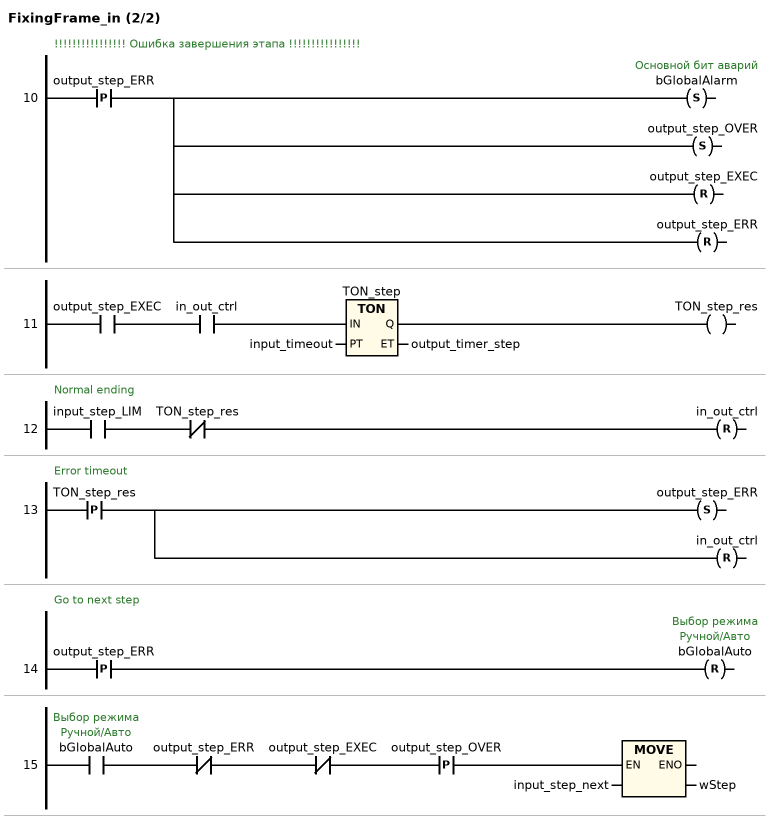
// NETWORK 10
// !!!!!!!!!!!!!!!! Ошибка завершения этапа !!!!!!!!!!!!!!!!
//   bGlobalAlarm: Основной бит аварий
_rt4(CLK := output_step_ERR);
bGlobalAlarm S= _rt4.Q;
output_step_OVER S= _rt4.Q;
output_step_EXEC R= _rt4.Q;
output_step_ERR R= _rt4.Q;

// NETWORK 11
TON_step(IN := output_step_EXEC AND in_out_ctrl, PT := input_timeout, ET => output_timer_step); // TON
TON_step_res := TON_step.Q;

// NETWORK 12
// Normal ending
in_out_ctrl R= input_step_LIM AND NOT TON_step_res;

// NETWORK 13
// Error timeout
_rt5(CLK := TON_step_res);
output_step_ERR S= _rt5.Q;
in_out_ctrl R= _rt5.Q;

// NETWORK 14
// Go to next step
//   bGlobalAuto: Выбор режима Ручной/Авто
_rt6(CLK := output_step_ERR);
bGlobalAuto R= _rt6.Q;

// NETWORK 15
//   bGlobalAuto: Выбор режима Ручной/Авто
_rt7(CLK := output_step_OVER);
IF bGlobalAuto AND NOT output_step_ERR AND NOT output_step_EXEC AND _rt7.Q THEN wStep := input_step_next; END_IF

END_PROGRAM

// MyController/Application/module_unites/FixingFrame_out
PROGRAM FixingFrame_out
VAR_INPUT
	input_step_INIT: BOOL;
	input_step_num: INT;
	input_step_LIM: BOOL;
	input_step_next: INT;
	input_timeout: TIME;
END_VAR

VAR_OUTPUT
	output_step_EXEC: BOOL;
	output_step_OVER: BOOL;
	output_step_ERR: BOOL;
	output_timer_step: TIME;
END_VAR
VAR_IN_OUT
	in_out_ctrl: BOOL;
END_VAR
VAR
	TON_step: TON;
	TON_step_res: BOOL;
	step_active: BOOL;
	TON_delay: TON;
	timer_delay: TIME;
	ton_delay_ok: BOOL;
END_VAR
VAR // added by the converter: edge detectors and wires of the graphical bodies
    _rt1, _rt2, _rt3, _rt4, _rt5, _rt6, _rt7 : R_TRIG;
    _w1, _w2 : BOOL;
    _ft1 : F_TRIG;
END_VAR

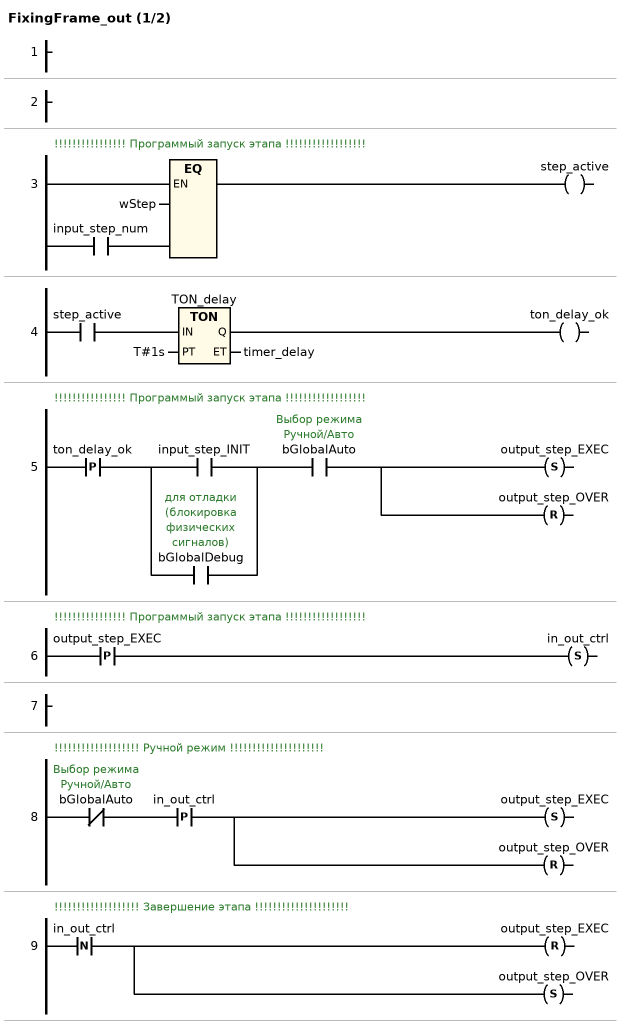
// NETWORK 1

// NETWORK 2

// NETWORK 3
// !!!!!!!!!!!!!!!! Программый запуск этапа !!!!!!!!!!!!!!!!!!
step_active := wStep = input_step_num;

// NETWORK 4
TON_delay(IN := step_active, PT := T#1s, ET => timer_delay); // TON
ton_delay_ok := TON_delay.Q;

// NETWORK 5
// !!!!!!!!!!!!!!!! Программый запуск этапа !!!!!!!!!!!!!!!!!!
//   bGlobalDebug: для отладки (блокировка физических сигналов)
//   bGlobalAuto: Выбор режима Ручной/Авто
_rt1(CLK := ton_delay_ok);
_w1 := _rt1.Q AND (input_step_INIT OR bGlobalDebug) AND bGlobalAuto;
output_step_EXEC S= _w1;
output_step_OVER R= _w1;

// NETWORK 6
// !!!!!!!!!!!!!!!! Программый запуск этапа !!!!!!!!!!!!!!!!!!
_rt2(CLK := output_step_EXEC);
in_out_ctrl S= _rt2.Q;

// NETWORK 7

// NETWORK 8
// !!!!!!!!!!!!!!!!!!! Ручной режим !!!!!!!!!!!!!!!!!!!!!
//   bGlobalAuto: Выбор режима Ручной/Авто
_rt3(CLK := in_out_ctrl);
_w2 := NOT bGlobalAuto AND _rt3.Q;
output_step_EXEC S= _w2;
output_step_OVER R= _w2;

// NETWORK 9
// !!!!!!!!!!!!!!!!!!! Завершение этапа !!!!!!!!!!!!!!!!!!!!!
_ft1(CLK := in_out_ctrl);
output_step_EXEC R= _ft1.Q;
output_step_OVER S= _ft1.Q;

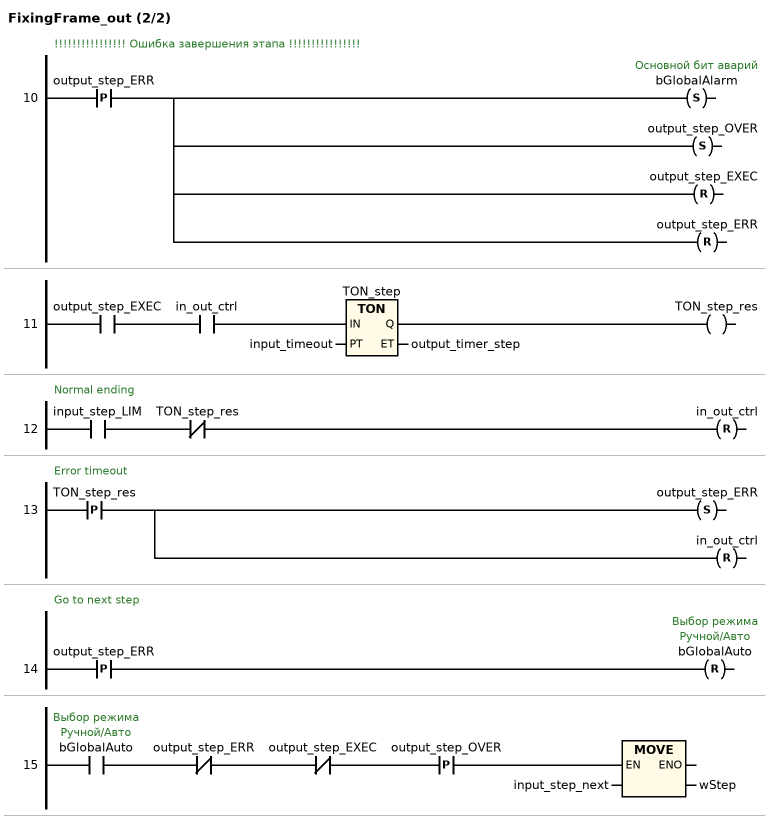
// NETWORK 10
// !!!!!!!!!!!!!!!! Ошибка завершения этапа !!!!!!!!!!!!!!!!
//   bGlobalAlarm: Основной бит аварий
_rt4(CLK := output_step_ERR);
bGlobalAlarm S= _rt4.Q;
output_step_OVER S= _rt4.Q;
output_step_EXEC R= _rt4.Q;
output_step_ERR R= _rt4.Q;

// NETWORK 11
TON_step(IN := output_step_EXEC AND in_out_ctrl, PT := input_timeout, ET => output_timer_step); // TON
TON_step_res := TON_step.Q;

// NETWORK 12
// Normal ending
in_out_ctrl R= input_step_LIM AND NOT TON_step_res;

// NETWORK 13
// Error timeout
_rt5(CLK := TON_step_res);
output_step_ERR S= _rt5.Q;
in_out_ctrl R= _rt5.Q;

// NETWORK 14
// Go to next step
//   bGlobalAuto: Выбор режима Ручной/Авто
_rt6(CLK := output_step_ERR);
bGlobalAuto R= _rt6.Q;

// NETWORK 15
//   bGlobalAuto: Выбор режима Ручной/Авто
_rt7(CLK := output_step_OVER);
IF bGlobalAuto AND NOT output_step_ERR AND NOT output_step_EXEC AND _rt7.Q THEN wStep := input_step_next; END_IF

END_PROGRAM

// MyController/Application/HiddenPOU
FUNCTION HiddenPOU : BOOL

VAR_INPUT
	pHiddenFunc: POINTER TO WORD;
END_VAR
VAR
	pRead: POINTER TO BYTE;
	pWrite: POINTER TO BYTE;
END_VAR

pRead := pHiddenFunc + 400;
pWrite := pHiddenFunc + 4400;
HiddenPOU := TRUE;

END_FUNCTION
